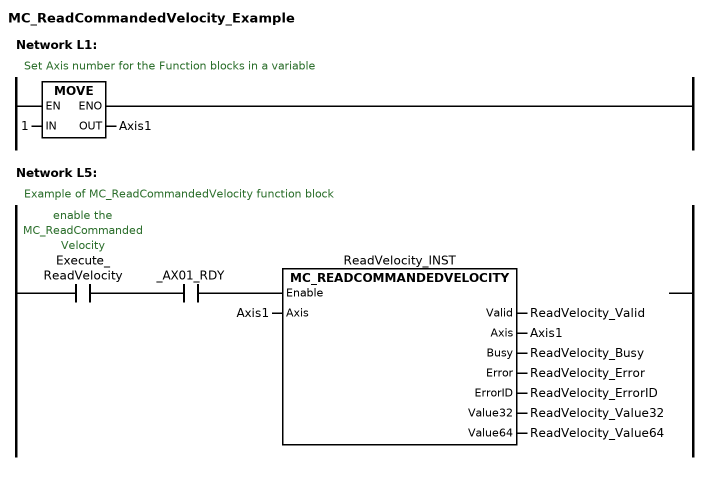
(* [picture p24: MC_ReadCommandedVelocity_Example rungs L1-L5] *)
(* Set Axis number for the Function blocks in a variable *)
(* Rung L1 *)
Axis1 := 1;
(* Example of MC_ReadCommandedVelocity function block *)
(* Rung L5 *)
ReadVelocity_INST(Enable := Execute_ReadVelocity AND _AX01_RDY, Axis := Axis1, Valid => ReadVelocity_Valid, Axis => Axis1, Busy => ReadVelocity_Busy, Error => ReadVelocity_Error, ErrorID => ReadVelocity_ErrorID, Value32 => ReadVelocity_Value32, Value64 => ReadVelocity_Value64);
END_PROGRAM

PROGRAM MC_ReadCommandedTorque_Example (* task: Scan Program *)
(* example of MC_ReadCommandedTorque function block *)
VAR
    Axis1 : UINT; (* used to tell MC function blocks to use axis 1 *)
    Execute_ReadTorque : BOOL; (* enable MC_ReadCommandedTorque *)
    ReadTorque_Busy : BOOL; (* Busy status of MC_ReadCommandedTorque *)
    ReadTorque_Error : BOOL; (* error status of MC_ReadCommandedTorque *)
    ReadTorque_ErrorID : WORD; (* error identification for MC_ReadCommandedTorque *)
    ReadTorque_INST : MC_READCOMMANDEDTORQUE; (* MC_ReadCommandedTorque function block *)
    ReadTorque_Valid : BOOL; (* valid status of MC_ReadCommandedTorque *)
    ReadTorque_Value32 : REAL; (* REAL value of MC_ReadCommandedTorque *)
    ReadTorque_Value64 : LREAL; (* LREAL value for MC_ReadCommandedTorque *)
END_VAR

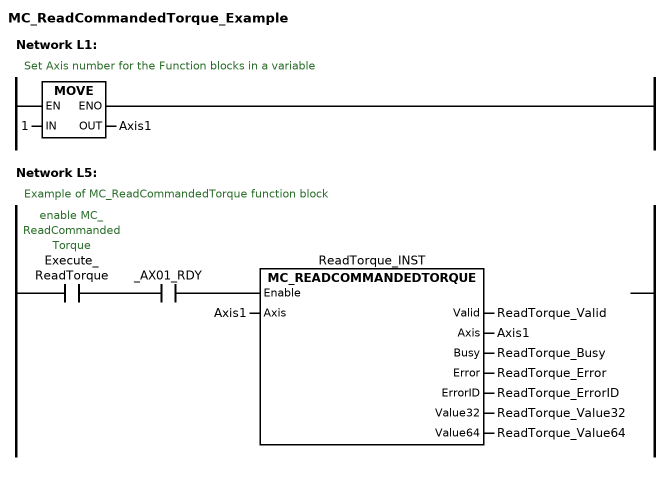
(* Set Axis number for the Function blocks in a variable *)
(* Rung L1 *)
Axis1 := 1;
(* Example of MC_ReadCommandedTorque function block *)
(* Rung L5 *)
ReadTorque_INST(Enable := Execute_ReadTorque AND _AX01_RDY, Axis := Axis1, Valid => ReadTorque_Valid, Axis => Axis1, Busy => ReadTorque_Busy, Error => ReadTorque_Error, ErrorID => ReadTorque_ErrorID, Value32 => ReadTorque_Value32, Value64 => ReadTorque_Value64);
END_PROGRAM